Staubli VAL3: onBackEvent.pgx

program onBackEvent(bool& x_bSave[] (dimensions=1))
  local num i
  local string l_sMessage[3]
  local num l_nLocal
  local bool l_bYes
  local string l_sAction[3]
  local num l_nIndex
  local string l_sButton[2]
  local TrajectoryItem l_tTraj
begin
  //
  // NB sEvent is the selected
  // element in the LIST
  //
  if nIndex!=0
    l_nIndex=nIndex-nUserItem
  else
    // change the name
    call changePoint(0)
  endIf
  if (l_nIndex)>0
    //
    //  There are 7 fields,
    //
    //
    call trajType:getTrajItem(l_tTraj,nIndexItem)
    switch l_nIndex
      case 1
        //
        //  change the movetype
        //
      break
      case 2
        //
        //  change the speed
        //
      break
      case 3
        //
        //  change the acceleration
        //
      break
      case 4
        //
        //  put a stop, after the robot reach to the point
        //
        // CLEAR THE STOP
        l_tTraj.toStop=false
      break
      case 5
        //
        //  set the blend (joint/off) for the point
        //
        l_tTraj.nom_speed.blend=off
      break
      case 6
        //
        // set TCP ON/OFF
        //
        // SET TCP OFF
        l_tTraj.nTcpAction=0
      break
      case 7,8,9
        //
        //  Delete the instruction
        //
        if l_tTraj.iInstr[l_nIndex-7].sType!=""
          call language:message(l_sMessage,171)
          call language:getYesNo(l_sButton)
          // ask the yes_no question
          call use:yes_no(l_sMessage,l_sButton,l_bYes)
          if l_bYes
            l_tTraj.iInstr[l_nIndex-7].sType=""
            l_tTraj.iInstr[l_nIndex-7].sData=""
          endIf
        endIf
      break
      case 10
        //
        //  set the distance from the point where the call will be actived
        //
        l_tTraj.distance=0
      break
    endSwitch
    //set and exit
    x_bSave=true
    call trajType:setTrajItem(l_tTraj,nIndexItem)
    call buildList()
  endIf
end
